# EPICS substitutions: apps/caenHvApp/Db/subs/HVBBHODO.substitutions
#
#This file will be eventuall autogenerated
file "db/caenhv.db" {
	pattern { Cr,   CrName,    CrType, Sl,   Ch,   Sys,  Det,    Element,       CScode, pwonoff, v0set,  i0set,   trip,    rampup,  rampdn, svmax,   enable}
		{"00", "BBTH-HV", "1527", "00", "00", "HV", "HODO", "101_L", "#C0",  "S2816",  "S512",  "S1280",  "S2560",   "S1024", "S768",   "S3328", "S256"}
		{"00", "BBTH-HV", "1527", "00", "01", "HV", "HODO", "201_L", "#C0",  "S2817", "S513", "S1281", "S2561", "S1025", "S769", "S3329", "S257" }
}
